TYPE udt_ECATNodeData_20221507 :
STRUCT
	NodeName:ARRAY[0..63] OF STRING;
	NodeType:ARRAY[0..63] OF STRING;
	State: ARRAY[0..63] OF UINT;
	TotalNodes:INT;
END_STRUCT
END_TYPE

(* stored: Version 1.1.0.1, ProductVersion 3.1.4024.11
   DUT udt_ECATNodeData_20221507: Id {a969ee17-2c67-4830-80df-d334ba38663d} *)
